(* Logix 5000 project; controller Process_Output Emulate 5570 rev 36.11; software revision 36.00 *)

TASK MainTask (continuous, watchdog 500 ms) : MainProgram

MODULES
   Local : Emulate 5570 (ICP 2, rev 36.11)
       : 1756-IB16 (ICP 3, rev 3.1, Input RPI 20 ms)
       : vendor 1 type 7 code 16 (ICP 4, rev 3.1, Output RPI 20 ms)
END_MODULES

VAR_GLOBAL   (* controller tags *)
   PROCESS_OUTPUT : ALIAS FOR Local:4:O.Data.0;   // Process Output
   SW_START : ALIAS FOR Local:3:I.Data.0;   // START Momentary N.O. Pushbutton
END_VAR

PROGRAM MainProgram   (* main routine FuncRoutine *)
VAR
   A_MATERIAL_MULTIPLIER : REAL;   // Material A Multiplier
   B_MATERIAL_MULTIPLIER : REAL;   // Material B Multiplier
   BAND_01 : FBD_BOOLEAN_AND := (In1 := 1, In2 := 1, In3 := 1, In4 := 1, In5 := 1, In6 := 1, In7 := 1, In8 := 1);
   BNOT_01 : FBD_BOOLEAN_NOT := (In := 1);
   BOR_01 : FBD_BOOLEAN_OR;
   C_MATERIAL_MULTIPLIER : REAL;   // Material C Multiplier
   D_MATERIAL_MULTIPLIER : REAL;   // Material D Multiplier
   HMI_NUM_SHEET : INT;   // Number of Material Sheets
   HMI_TYPE_SHEET : INT;   // Type of Sheets
   MATERIAL_MULTI_VALUE : REAL;   // Material Multiplier Value
   MUL_01 : FBD_MATH;
   MUL_03 : FBD_MATH;
   MUX_01 : MULTIPLEXER;
   TONR_01 : FBD_TIMER;
END_VAR

ROUTINE FuncHMI   (* function block diagram *)
   SHEET 1
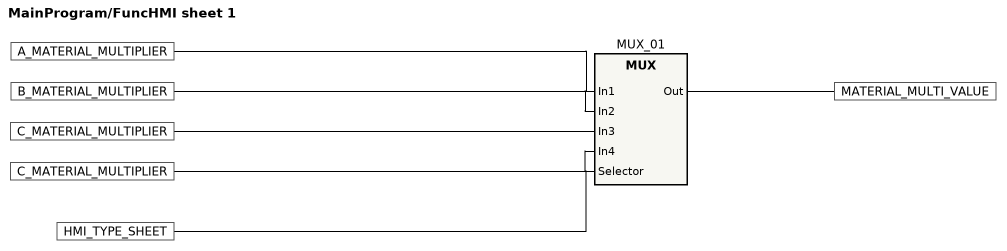
   MUX_01 : MUX(In1 := A_MATERIAL_MULTIPLIER, In2 := B_MATERIAL_MULTIPLIER, In3 := C_MATERIAL_MULTIPLIER, In4 := C_MATERIAL_MULTIPLIER, Selector := HMI_TYPE_SHEET);
   MATERIAL_MULTI_VALUE := MUX_01.Out;
END_ROUTINE

ROUTINE FuncRoutine   (* function block diagram *)
   SHEET 1
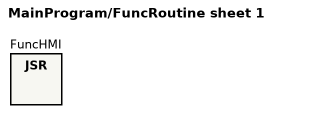
   FuncHMI : JSR();
   SHEET 2
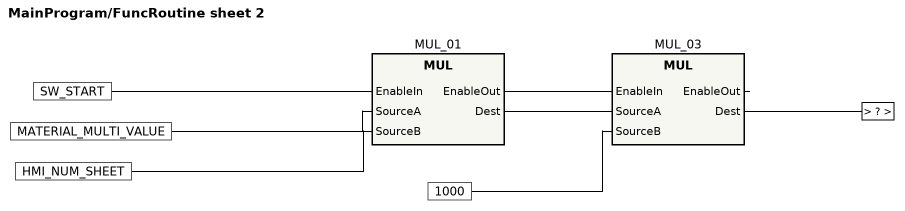
   MUL_01 : MUL(EnableIn := SW_START, SourceA := MATERIAL_MULTI_VALUE, SourceB := HMI_NUM_SHEET);
   MUL_03 : MUL(EnableIn := MUL_01.EnableOut, SourceA := MUL_01.Dest, SourceB := 1000);   // unwired pins: EnableOut
   WIRE(?) := MUL_03.Dest;
   SHEET 3
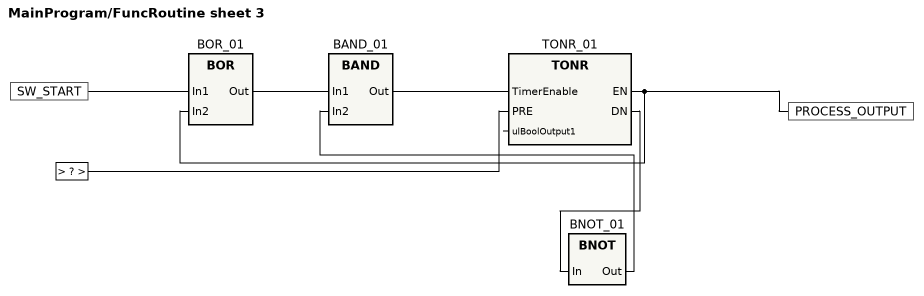
   BOR_01 : BOR(In1 := SW_START, In2 := TONR_01.EN {feedback});
   BNOT_01 : BNOT(In := TONR_01.DN {feedback});
   BAND_01 : BAND(In1 := BOR_01.Out, In2 := BNOT_01.Out);
   TONR_01 : TONR(TimerEnable := BAND_01.Out, PRE := WIRE(?));   // unwired pins: ulBoolOutput1
   PROCESS_OUTPUT := TONR_01.EN;
END_ROUTINE
END_PROGRAM
